FUNCTION_BLOCK FB_TrafficLight_Test EXTENDS TcUnit.FB_TestSuite
VAR
END_VAR

NewLightStartsInRed();
RedLightGoesGreenOnRequest();

METHOD PRIVATE NewLightStartsInRed
VAR
	light       : FB_TrafficLight;
    actualState : E_LightState;
END_VAR
TEST('NewLightStartsInRed');

actualState := light.CurrentState;   // read the property into a variable first

AssertEquals_INT(
    Expected := TO_INT(E_LightState.Red),
    Actual   := TO_INT(actualState),
    Message  := 'A new light should start in RED');

TEST_FINISHED();
END_METHOD

METHOD PRIVATE RedLightGoesGreenOnRequest
VAR
	light       : FB_TrafficLight;
    actualState : E_LightState;
END_VAR
TEST('RedLightGoesGreenOnRequest');

// light starts in Red (verified by the previous test)
light.RequestGreen();             
actualState := light.CurrentState;

AssertEquals_INT(
    Expected := TO_INT(E_LightState.Green),
    Actual   := TO_INT(actualState),
    Message  := 'A light in RED should go GREEN when requested');

TEST_FINISHED();
END_METHOD

END_FUNCTION_BLOCK

(* stored: Version 1.1.0.1, ProductVersion 3.1.4024.12
   POU FB_TrafficLight_Test: Id {05a59aff-e522-47ed-8604-19fdd813a76a}, SpecialFunc None
   Method NewLightStartsInRed: Id {870cd3fb-b52e-4f56-bf23-b9ba4841ad63}
   Method RedLightGoesGreenOnRequest: Id {9ffbc1b8-7f1c-42d9-ad91-886f75c1297d} *)
